Fanuc KAREL source: kt00006.KL

-- PROVISIONAL review KL for V940-1; original PC SHA256 965331df3aaf398be92bfafe7849428af16ada811f9d60ba7662376e6d3c0fe7
-- Incomplete behavior may be omitted. Consult companion uncertainty JSON. Do not deploy.
PROGRAM KT00006
%NOLOCKGROUP
VAR
  I1 : INTEGER
  OUT : REAL
-- UNRESOLVED_DECL Y2 type=002018
BEGIN
  -- V9_ZERO_TABLE_METADATA_HINT layout=0001; no indexed target words; source/name/runtime held
  -- UNRESOLVED_PC offsets 5-16; opcodes 2E,23
  -- UNRESOLVED_PC offsets 21-35; opcodes 2E,22,9D,33,B2
  -- UNRESOLVED_PC offsets 40-63; opcodes 21,22,9D,33,B1,52,64,23
  -- UNRESOLVED_PC offsets 68-72; opcodes 7F
END KT00006
